// TIA Portal project "babu_RisingEdgeV19" (V19)

(* hardware
DEVICE "S7-1200 station_1"  S7-1200 Station
   slot 0: "Rack_0"  S7-1200 Rack  Rack  V1.0
   slot 1: "PLC_1"  CPU 1212C DC/DC/DC  6ES7 212-1AE40-0XB0  V4.6
*)

// ===== PLC "PLC_1"  CPU 1212C DC/DC/DC =====

VAR_GLOBAL   // PLC tag table "Default tag table"
   "IP1" AT %M0.0 : Bool;
   "MEM" AT %M0.1 : Bool;
   "OP1" AT %Q0.0 : Bool;
   "OP1MEM" AT %M0.2 : Bool;
END_VAR

ORGANIZATION_BLOCK "Main"   // OB1, LAD, ProgramCycle
TITLE = "Main Program Sweep (Cycle)"
{ S7_Optimized_Access := 'TRUE' }
VERSION : 0.1
   VAR_INPUT
      Initial_Call : Bool;   // Initial call of this OB
      Remanence : Bool;   // =True, if remanent data are available
   END_VAR
   VAR_TEMP   // added for the SCL form of the ladder/FBD networks
      _w1 : Bool;
   END_VAR
BEGIN

REGION Network 1
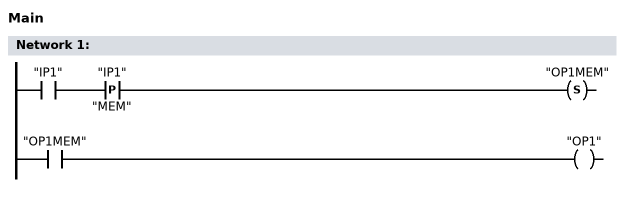
   RUNG wire#powerrail
      Contact( "IP1" )
      P_Contact(operand := "IP1", bit := "MEM")
      S_Coil( "OP1MEM" )
   END_RUNG
   RUNG wire#powerrail
      Contact( "OP1MEM" )
      Coil( "OP1" )
   END_RUNG
   // the same network as SCL:
   #_w1 := "IP1" AND "IP1" AND NOT "MEM";   // rising edge of "IP1"
   "MEM" := "IP1";
   IF #_w1 THEN "OP1MEM" := TRUE; END_IF;
   "OP1" := "OP1MEM";
END_REGION
END_ORGANIZATION_BLOCK